FUNCTION_BLOCK FB_TestElementDensity EXTENDS TcUnit.FB_TestSuite
VAR
	fbElementDensity : FB_ElementDensity;
END_VAR

TEST('fbElementDensity Si lookup');

fbElementDensity(sName:='Si');
AssertTrue(fbElementDensity.bFound, 'Silicon not found');
AssertEquals_LREAL(2.33, fbElementDensity.fValue, Delta:=0.0001, Message:='Element density constant value');
TEST_FINISHED();

TEST('fbElementDensity bad name lookup');
fbElementDensity(sName:='Silicon');
AssertFalse(fbElementDensity.bFound, 'Silicon should not be found');
AssertEquals_LREAL(0.0, fbElementDensity.fValue, Delta:=0.0001, Message:='Element density constant value');
TEST_FINISHED();

END_FUNCTION_BLOCK

(* stored: Version 1.1.0.1, ProductVersion 3.1.4022.18
   POU FB_TestElementDensity: Id {261ac554-92a7-43d8-87eb-033d058900e2}, SpecialFunc None *)
